FUNCTION_BLOCK FB_CRYO_SENSOR_BASE
VAR_INPUT
END_VAR
VAR
	{attribute 'OPC.UA.DA' := '0'}
	i_nStatus	AT %I*: UINT;
	{attribute 'OPC.UA.DA' := '0'}
	i_nValue	AT%I*:	INT;
	
	{attribute 'OPC.UA.DA' := '0'}
	bStarted:		BOOL := FALSE;
	{attribute 'OPC.UA.DA' := '0'}
	toggleTimer:	TON;		// Timer for PDO (alive) toggle
	{attribute 'OPC.UA.DA' := '0'}
	toggleTrig:		R_TRIG;		// PDO (alive) toggle detection
	
	RefStat: 	REFERENCE TO T_CRYO_SENSOR_STATUS;
END_VAR

// Get the raw reading and the status of the input channel
M_ReadSensor();

// Calculate value and validity
M_SetStatus();

// Get input channel status and the raw reading
METHOD M_ReadSensor
VAR_INPUT
END_VAR
// Get input channel status
RefStat.bInputUnder	:= (i_nStatus AND 2#0000_0000_0000_0001) <> 0;
RefStat.bInputOver	:= (i_nStatus AND 2#0000_0000_0000_0010) <> 0;
RefStat.bInputError	:= (i_nStatus AND 2#0000_0000_0100_0000) <> 0;
RefStat.bInputToggle:= (i_nStatus AND 2#1000_0000_0000_0000) <> 0;
RefStat.bInputValid	:= (i_nStatus AND 2#0100_0000_0000_0000)  = 0;	// 0 -> PDO OK

// Get the raw reading
RefStat.nRawValue	:= i_nValue;

//
// Check if the terminal is alive.
// Start the time that will expire in 3 sec.
// If bToggle bit triggers before the timer expires, 
// this is the sign that the terminal is alive.
//
IF NOT bStarted THEN
	bStarted	:= TRUE;
	toggleTimer(IN:=FALSE);
END_IF
toggleTimer(IN:=TRUE,PT:=T#3S);
toggleTrig(CLK:=RefStat.bInputToggle);

IF toggleTrig.Q THEN
	// bToggle bit has triggered. Terminal is alive.
	RefStat.bInputActive	:= TRUE;
	// Restart the timer
	toggleTimer(IN:=FALSE);
ELSIF toggleTimer.Q THEN
	// bInputToggle bit has not triggered within 3 sec. Terminal is NOT alive.
	RefStat.bInputActive	:= FALSE;
	// Restart the timer
	toggleTimer(IN:=FALSE);
END_IF
END_METHOD

METHOD M_SetStatus
VAR_INPUT
END_VAR
// TODO USER: Implement the method.
END_METHOD

END_FUNCTION_BLOCK

(* stored: Version 1.1.0.1, ProductVersion 3.1.4024.3
   POU FB_CRYO_SENSOR_BASE: Id {c37197f1-7325-44a1-a2c9-824a796d0c57}, SpecialFunc None
   Method M_ReadSensor: Id {af917b5a-b58d-4cde-9881-8b0f43d46c6f}
   Method M_SetStatus: Id {32db71e3-1ed5-4278-a637-97edbf1d9e83} *)
